FUNCTION_BLOCK FB_NormalWash IMPLEMENTS I_WashStrategy
VAR
	stWashSettings : ST_WashSettings;
END_VAR

METHOD FB_init : BOOL
VAR_INPUT
	bInitRetains : BOOL; // if TRUE, the retain variables are initialized (warm start / cold start)
	bInCopyCode : BOOL;  // if TRUE, the instance afterwards gets moved into the copy code (online change)
END_VAR
IF stWashSettings.sDescription = '' THEN
	stWashSettings.rWashTemperature := GVL_WashConstants.NORMAL_TEMP;
	stWashSettings.nSpinSpeed:= GVL_WashConstants.NORMAL_SPIN;
	stWashSettings.tWashDuration := GVL_WashConstants.NORMAL_WASH_TIME;
	stWashSettings.sDescription := GVL_WashConstants.NORMAL_DESC;
	
END_IF
FB_init :=TRUE;
END_METHOD

{warning 'add method implementation '}
METHOD GetProgramName : STRING
GetProgramName := 'Normal';
END_METHOD

METHOD GetRinseTime : TIME;
VAR_INPUT
END_VAR
GetRinseTime := GVL_WashConstants.INTENSIVE_WASH_RINSE_TIME;
END_METHOD

METHOD GetSpinTime : TIME
VAR_INPUT
END_VAR
GetSpinTime := GVL_WashConstants.INTENSIVE_WASH_SPIN_TIME;
END_METHOD


METHOD GetWashSettings : ST_WashSettings
GetWashSettings := stWashSettings;
END_METHOD

END_FUNCTION_BLOCK

(* stored: Version 1.1.0.1, ProductVersion 3.1.4024.16
   POU FB_NormalWash: Id {4501bad4-73b6-4180-bc5c-3147bcd1749d}, SpecialFunc None
   Method FB_init: Id {cca724aa-2f2f-40b8-a35f-a84be90a8aef}
   Method GetProgramName: Id {7f7c6360-78fe-436f-a4d1-1edf53ad730b}
   Method GetRinseTime: Id {5ade095b-1f78-4211-adac-0afdf8734c4c}
   Method GetSpinTime: Id {88de4e58-e819-4bbe-a1a5-d1e131a9edcf}
   Method GetWashSettings: Id {e376caec-c9b4-43e6-b724-82e3201f633c} *)
